FUNCTION_BLOCK PUBLIC FB_Info IMPLEMENTS I_Info
VAR_INPUT
END_VAR
VAR_OUTPUT
END_VAR
VAR
    sInstancePath:				REFERENCE TO STRING(255);
	eState:						REFERENCE TO E_State;
	fbReadSymInfo: 				PLC_ReadSymInfoByNameEx;
	nIndex:						DINT;
END_VAR
VAR_STAT
	nCycle: 					UDINT;
	nTimestamp: 				ULINT;
END_VAR

GETCURTASKINDEXEX(GETCURTASKINDEXEX => nIndex);
IF nCycle <> TwinCAT_SystemInfoVarList._TaskInfo[nIndex].CycleCount THEN
	nCycle:= TwinCAT_SystemInfoVarList._TaskInfo[nIndex].CycleCount;
	nTimestamp:= F_GetSystemTime();
END_IF

fbReadSymInfo(
	NETID:= , 
	PORT:= , 
	SYMNAME:= , 
	START:= , 
	TMOUT:= , 
	BUSY=> , 
	ERR=> , 
	ERRID=> , 
	SYMINFO=> , 
	OVTYPE=> , 
	OVCOMMENT=> );

METHOD FB_init : BOOL
VAR_INPUT
	bInitRetains : BOOL; // if TRUE, the retain variables are initialized (warm start / cold start)
	bInCopyCode : BOOL;  // if TRUE, the instance afterwards gets moved into the copy code (online change)
	sInstancePath:			REFERENCE TO STRING(255);
	eState:					REFERENCE TO E_State;
	
END_VAR
THIS^.sInstancePath REF= sInstancePath;
THIS^.eState REF= eState;
M_Initialize();
END_METHOD

METHOD PROTECTED M_Initialize
VAR_INPUT
END_VAR
VAR
    sName:				STRING(255);
    nPosition:			INT;
END_VAR
sName := CONCAT(TwinCAT_SystemInfoVarList._AppInfo.ProjectName, '.');

nPosition := FIND(sInstancePath, sName);
IF nPosition > 0 THEN
    fbReadSymInfo.SYMNAME:= DELETE(sInstancePath, nPosition-1 + LEN(sName), 1);
END_IF

nPosition := FIND(fbReadSymInfo.SYMNAME, sName);

IF nPosition > 0 THEN
    fbReadSymInfo.SYMNAME:= DELETE(fbReadSymInfo.SYMNAME, nPosition - 1 + LEN(sName), 1);
END_IF

fbReadSymInfo.PORT:= TwinCAT_SystemInfoVarList._AppInfo.AdsPort;
fbReadSymInfo.START:= TRUE;
END_METHOD

PROPERTY PUBLIC P_Class : String(255)
GET
P_Class:= fbReadSymInfo.SYMINFO.symDataType;
END_GET
END_PROPERTY

PROPERTY PUBLIC P_Comment : String(255)
GET
P_Comment:= fbReadSymInfo.SYMINFO.symComment;
END_GET
END_PROPERTY

PROPERTY PUBLIC P_Instance : String(255)
GET
P_Instance:= fbReadSymInfo.SYMNAME;
END_GET
END_PROPERTY

PROPERTY PUBLIC P_State : E_State
GET
P_State:= eState;
END_GET
END_PROPERTY

PROPERTY PUBLIC P_Timestamp : ULINT
GET
P_Timestamp:= nTimestamp;
END_GET
END_PROPERTY

END_FUNCTION_BLOCK

(* stored: Version 1.1.0.1
   POU FB_Info: Id {eea7efb5-6652-45a3-b451-b5b834049a65}, SpecialFunc None
   Method FB_init: Id {b3af4ade-e4ea-4784-b0ea-8fa1426af073}
   Method M_Initialize: Id {0b417d91-c3b8-4144-89a2-d1e8ea1316dd}
   Property P_Class: Id {149d54ac-7219-431b-bfce-ba7c9704ea45}
   Get Get: Id {740bc1cd-c684-4cda-ac0a-196c933124fe}
   Property P_Comment: Id {2f19e0ac-9ace-4998-a64c-c83a5e4179c9}
   Get Get: Id {65efe2d4-df35-4bc5-aec6-6947856bcef9}
   Property P_Instance: Id {9eb0e8a4-0ed9-4848-97b2-cb18e1840110}
   Get Get: Id {8d15c27d-b883-4397-bad1-a1acae195710}
   Property P_State: Id {c747533f-000a-4f36-b4ba-f00b2fbb73f7}
   Get Get: Id {88d67c77-472d-4a63-bef7-c9cec62b2136}
   Property P_Timestamp: Id {a51f1ff9-c398-4582-9d70-e288f1c0d28c}
   Get Get: Id {ca050bdc-7777-4205-b941-d6aa9ea30447} *)
